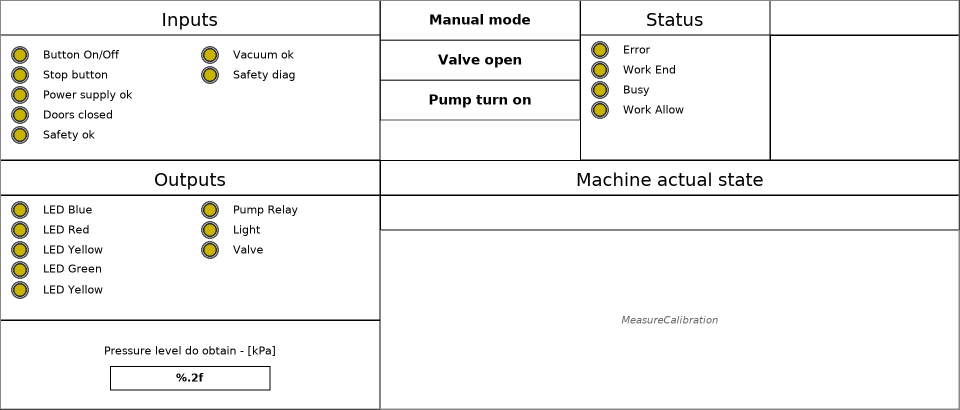
VISUALIZATION vUnderPressureFrame_V2  // 960x410
VAR_IN_OUT
	stInOuts : stUnderPressureTesterInOuts_V2;
	stParams : stUnderPressureTestParams_V2;
	stStatus	: stUnderPressureTestStatus_V2;
	iWorkStep	: INT;
END_VAR
    Rectangle (0,320 380x90)
    Rectangle (0,195 380x125)
    Rectangle (580,0 380x35)
    Lamp1 (10,45 20x20), variable: stInOuts.bSwitchOnOff, style: Lamp-Lamp1-Yellow
    Lamp1 (10,65 20x20), variable: stInOuts.bStopButtonNC, style: Lamp-Lamp1-Yellow
    Lamp1 (10,85 20x20), variable: stInOuts.bPhaseControlRelay, style: Lamp-Lamp1-Yellow
    Lamp1 (10,105 20x20), variable: stInOuts.bLockSens, style: Lamp-Lamp1-Yellow
    Lamp1 (10,125 20x20), variable: stInOuts.bSafetyOK, style: Lamp-Lamp1-Yellow
    Label (40,45 150x20), "Button On/Off"
    Label (40,65 150x20), "Stop button"
    Label (40,85 150x20), "Power supply ok"
    Label (40,105 150x20), "Doors closed"
    Label (40,125 150x20), "Safety ok"
    Rectangle (0,0 380x35)
    Label (0,5 380x30), "Inputs"
    Rectangle (380,0 200x40), "Manual mode", input disabled if: NOT GVL.fbUserLogin.bPermissionGranted
        OnMouseClick: toggle stStatus.bManual
    Rectangle (380,40 200x40), "Valve open", input disabled if: NOT GVL.fbUserLogin.bPermissionGranted
        OnMouseClick: toggle stInOuts.bEValve
    Rectangle (380,80 200x40), "Pump turn on", input disabled if: NOT GVL.fbUserLogin.bPermissionGranted
        OnMouseClick: toggle stInOuts.bPumpRly
    Rectangle (580,0 190x160)
    Rectangle (770,35 190x125)
    Label (580,5 190x30), "Status"
    Rectangle (0,160 380x35)
    Label (620,40 150x20), "Error"
    Lamp1 (590,40 20x20), variable: stStatus.bError, style: Lamp-Lamp1-Yellow
    Lamp1 (590,60 20x20), variable: stStatus.bWorkEnd, style: Lamp-Lamp1-Yellow
    Lamp1 (590,80 20x20), variable: stStatus.bBusy, style: Lamp-Lamp1-Yellow
    Label (620,60 150x20), "Work End"
    Label (620,80 150x20), "Busy"
    Label (40,200 150x20), "LED Blue"
    Lamp1 (10,200 20x20), variable: stInOuts.bLEDBlue, style: Lamp-Lamp1-Yellow
    Lamp1 (10,220 20x20), variable: stInOuts.bLEDRed, style: Lamp-Lamp1-Yellow
    Lamp1 (10,240 20x20), variable: stInOuts.bLEDYellow, style: Lamp-Lamp1-Yellow
    Label (40,220 150x20), "LED Red"
    Label (40,240 150x20), "LED Yellow"
    Label (230,200 150x20), "Pump Relay"
    Lamp1 (200,200 20x20), variable: stInOuts.bPumpRly, style: Lamp-Lamp1-Yellow
    Lamp1 (200,220 20x20), variable: stInOuts.bLight, style: Lamp-Lamp1-Yellow
    Lamp1 (200,240 20x20), variable: stInOuts.bEValve, style: Lamp-Lamp1-Yellow
    Label (230,220 150x20), "Light"
    Label (230,240 150x20), "Valve"
    Label (380,165 580x30), "Machine actual state"
    Rectangle (380,160 580x35)
    Rectangle (380,195 580x35), text list: 'tlVacuumStep_V2', text index: iWorkStep
    Lamp1 (200,45 20x20), variable: stInOuts.bVaccumOK, style: Lamp-Lamp1-Yellow
    Lamp1 (200,65 20x20), variable: stInOuts.bSafetyDiag, style: Lamp-Lamp1-Yellow
    Label (230,45 150x20), "Vacuum ok"
    Label (230,65 150x20), "Safety diag"
    Label (0,165 380x30), "Outputs"
    Lamp1 (10,280 20x20), variable: stInOuts.bLEDGreen, style: Lamp-Lamp1-Yellow
    Lamp1 (10,260 20x20), variable: stInOuts.bLEDGreen, style: Lamp-Lamp1-Yellow
    Label (40,259 150x20), "LED Green"
    Label (40,280 150x20), "LED Yellow"
    Lamp1 (590,100 20x20), variable: stStatus.bWorkAllow, style: Lamp-Lamp1-Yellow
    Label (620,100 150x20), "Work Allow"
    Rectangle (110,366 160x24), "%.2f", text variable: stParams.rVaccumLevelToObtain, input disabled if: NOT GVL.fbUserLogin.bPermissionGranted
        OnMouseClick: write the text variable via Default, format %d
    Label (100,341 180x20), "Pressure level do obtain - [kPa]"
    Frame (380,230 580x180), input disabled if: NOT GVL.fbUserLogin.bPermissionGranted
        shows MeasureCalibration(stMeasureData := stParams.stVacuumData, diAnalogIn := stInOuts.iVacuumLevel, MeasureName := 'Vacuum calibration')
    Rectangle (0,0 380x160)
END_VISUALIZATION

(* stored: Version 1.1.0.1, ProductVersion 3.1.4024.13
   Visu vUnderPressureFrame_V2: Id {8f0471dc-743f-4db4-a056-6ec812b0507c} *)
